// TIA Portal V20 export
FUNCTION "StepToString" : String   // FC86, SCL
// stored: Namespace Unit1.Em3, SetENOAutomatically false
   VAR_INPUT
      StepDINT : DInt;   // DINT value of the step
   END_VAR
BEGIN
   // Translates the sequence step number to the step name
   // Adjusted for Sequence_1_WebGuid real use case

   CASE #StepDINT OF
       1:
           #StepToString := 'Idle';

       101:
           #StepToString := 'JOB[1] Condition';
       111:
           #StepToString := 'Web Guide EPC Mode Check';
       121:
           #StepToString := 'Electro Pneumatic Regulator Check';
       131:
           #StepToString := 'Dancer WorkPos Command';
       141:
           #StepToString := 'Dancer Encoder Check';
       191:
           #StepToString := 'JOB[1] Step End';

       901:
           #StepToString := 'Immediate Stop';

       ELSE
           #StepToString := 'N/A';

   END_CASE;
END_FUNCTION
